(* PLC project Unnamed, Unknown Unnamed 1 *)
(* stored: creationDateTime 2025-11-05T12:12:45, modificationDateTime 2025-11-05T15:01:02 *)

TYPE MotorStruct : STRUCT
  Running : BOOL := False;
  SafeTemp : BOOL := True;
END_STRUCT;
END_TYPE

PROGRAM main
  VAR_EXTERNAL
    PB1 : BOOL;  (* Hardware Input *)
    PB2 : BOOL;  (* Hardware Input *)
    PB3 : BOOL;  (* Hardware Input *)
    PB4 : BOOL;  (* Hardware Input *)
    AI_TempSensor : REAL;  (* Hardware Input *)
    MotorState : MotorStruct;  (* Struct for other Programs to monitor motor state *)
  END_VAR
  VAR
    StartButton : BOOL := False;  (* Start button logic state *)
    StopButton : BOOL := True;  (* Stop button logic state *)
    EStopButton : BOOL := True;  (* EStop button logic state *)
    M_Temp : REAL;  (* Local temperature reading *)
    Safe : BOOL := True;  (* Is motor safe to run *)
    M_Sart : BOOL := False;  (* Command Trigger *)
    M_Running : BOOL := False;  (* Motor Running State *)
    Fault_MotorTemp : BOOL := False;  (* Fault for motor overheating *)
    FaultMotorTemp_Reset : BOOL := False;  (* Reset for fault state *)
  END_VAR

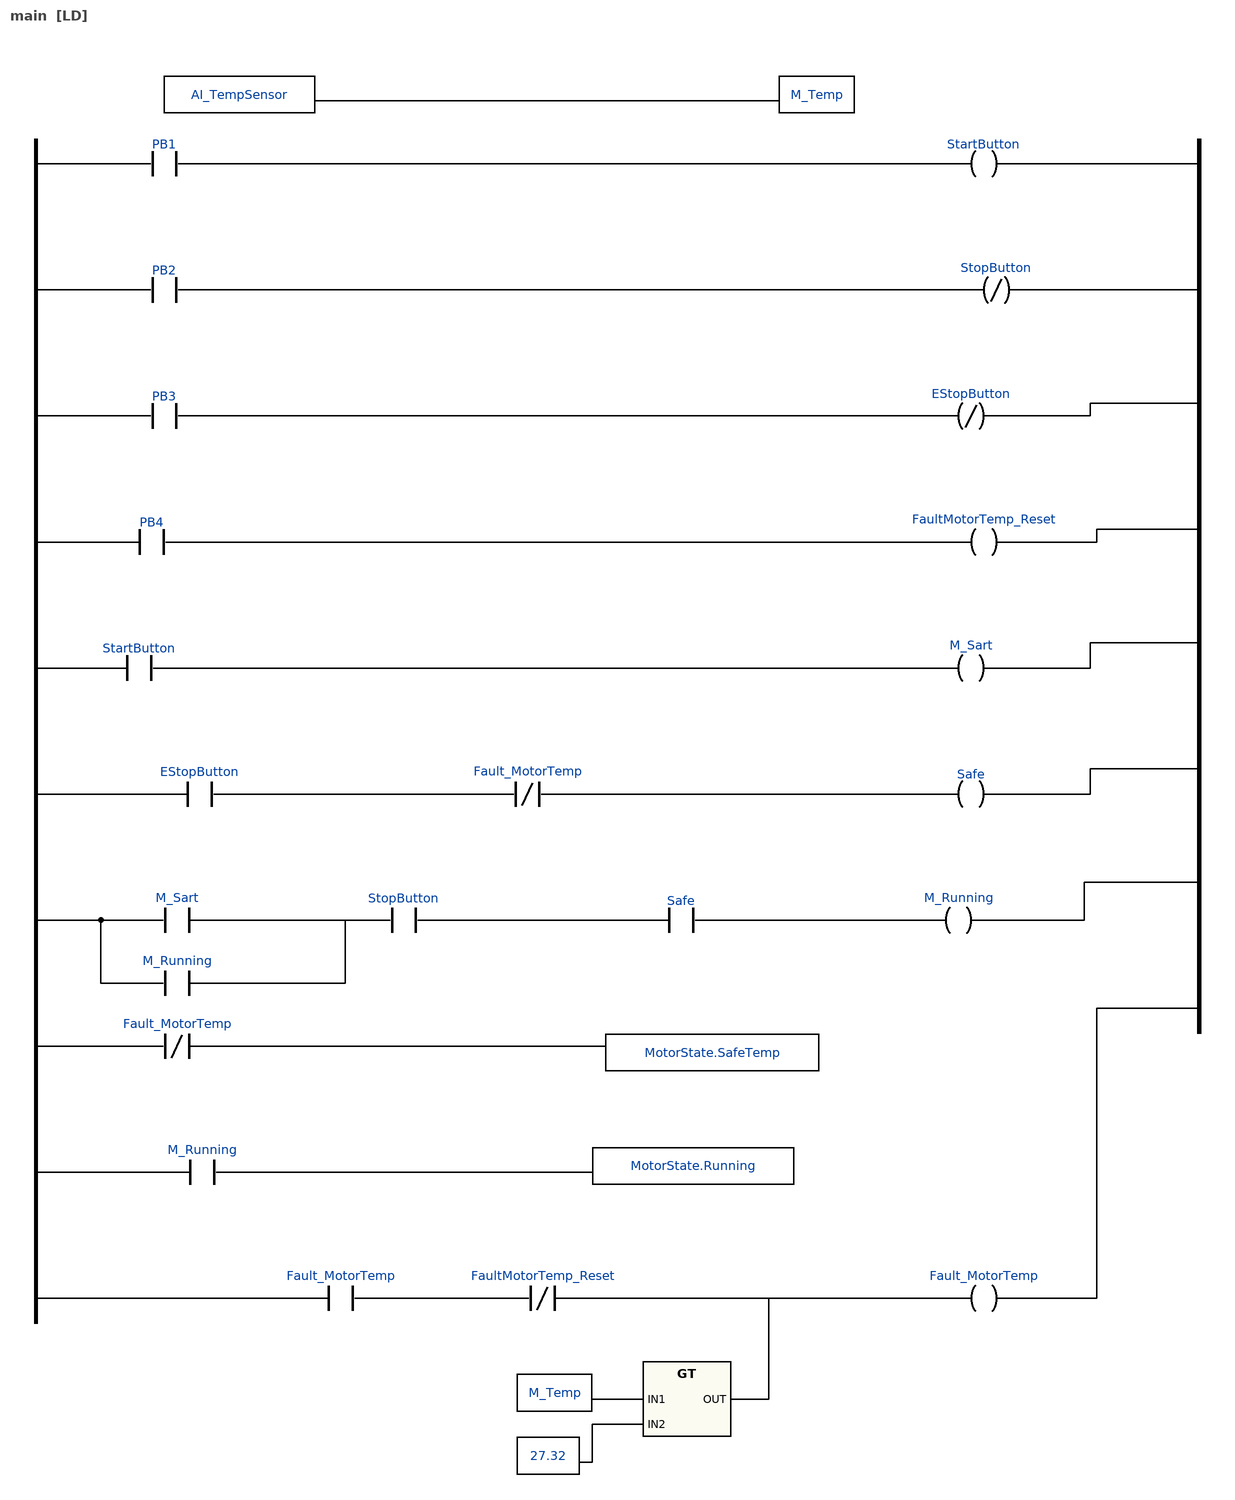
(* LD diagram, written out as Structured Text *)
StartButton := PB1;
StopButton := NOT PB2;
EStopButton := NOT PB3;
M_Temp := AI_TempSensor;
M_Running := (M_Sart OR M_Running) AND StopButton AND Safe;
Fault_MotorTemp := M_Temp > 27.32 OR Fault_MotorTemp AND NOT FaultMotorTemp_Reset;
Safe := EStopButton AND NOT Fault_MotorTemp;
MotorState.Running := M_Running;
MotorState.SafeTemp := NOT Fault_MotorTemp;
M_Sart := StartButton;
FaultMotorTemp_Reset := PB4;
END_PROGRAM

CONFIGURATION Config0
  VAR_GLOBAL
    PB1 AT %IX0.0 : BOOL := False;  (* The Start Push Button *)
    PB2 AT %IX0.1 : BOOL := False;  (* The Stop Push Button *)
    PB3 AT %IX0.2 : BOOL := False;  (* The Emergency Stop Push button *)
    PB4 AT %IX0.3 : BOOL := False;  (* Reset Motor Fault *)
    AI_TempSensor AT %IX0.4 : REAL := 0.0;  (* Temperature Sensor for the Motor *)
    MotorState : MotorStruct;
  END_VAR
  RESOURCE Res0 ON PLC
    TASK task0(INTERVAL := T#20ms, PRIORITY := 0);
    PROGRAM instance0 WITH task0 : main;
  END_RESOURCE
END_CONFIGURATION
